TYPE ST_RejectReason_PK4_OUT2 :
STRUCT
	Reason	:STRING;
END_STRUCT
END_TYPE

(* stored: Version 1.1.0.1, ProductVersion 3.1.4024.13
   DUT ST_RejectReason_PK4_OUT2: Id {46dfe178-7b17-45ec-8f11-a33189b61a9d} *)
